Staubli VAL3: strfillchr.pgx

public program strFillChr(string x_sIn, string& x_sOut[], string x_sChar)
  local num l_nIndex
begin
  //-----------------------------------------------------------------------
  //Header begin
  //Description of program
  //  To fill the string with custom characters.
  //  Usually using for a cryptage.
  //
  //Input parameters
  //  string x_sIn :
  //    role : string that you want modified
  //  string x_sChar :
  //    role : characters that you want replaced.
  //
  //Output parameters
  //  string x_sOut :
  //    role : string modified
  //
  //Example
  //   password cryptage
  //   call strFillChr(lPassword,lView,"*")
  //
  //History
  //  Creation : 28-04-08 - f.Rob
  //Header end
  //-----------------------------------------------------------------------
  x_sOut=""
  if getDisplayLen(x_sIn)>0
    for l_nIndex=0 to (getDisplayLen(x_sIn)-1)
      x_sOut=x_sOut+x_sChar
    endFor
  endIf
end
